// TIA Portal V19 export
DATA_BLOCK "MC_Home_DB"   // DB3
// stored: InstanceOfName MC_Home, OfSystemLibElement MC_Home, OfSystemLibVersion 7.0
"MC_Home"
   // VAR_INPUT
   //    Axis : TO_Axis;
   //    Execute : Bool;
   //    Position : Real;
   //    Mode : Int;
   // END_VAR
   // VAR_OUTPUT
   //    Done : Bool;
   //    Busy : Bool;
   //    CommandAborted : Bool;
   //    Error : Bool;
   //    ErrorID : Word;
   //    ErrorInfo : Word;
   //    ReferenceMarkPosition : Real;
   // END_VAR
   // VAR
   //    FB_ID : DInt;
   // END_VAR
BEGIN
END_DATA_BLOCK
